// TIA Portal project "Rectz" (V13)

(* hardware
DEVICE "S7300/ET200M station_1"  S7-300 station
   slot 0: "Rail_0"  Rail  6ES7 390-1***0-0AA0
   slot 1: "PS 307 5A_1"  PS 307 5A  6ES7 307-1EA01-0AA0
   slot 2: "PLC_1"  CPU 314C-2 PN/DP  6ES7 314-6EH04-0AB0  V3.3
      slot 2: "PROFINET interface_1"  PN-IO
         slot 1: "Port_1"  Port
         slot 2: "Port_2"  Port
      slot 5: "DI 24/DO 16_1"  DI24/DO16
      slot 6: "AI 5/AO 2_1"  AI5/AO2
      slot 7: "Count_1"  Counter
      slot 8: "Positioning_1"  Positioning
*)

// ===== PLC "PLC_1"  CPU 314C-2 PN/DP =====

VAR_GLOBAL   // PLC tag table "Default tag table"
   "Start" AT %I0.1 : Bool;   // Botão de start
   "Reset" AT %I0.2 : Bool;   // Botão de reset
   "Stop" AT %I0.3 : Bool;   // Botão de stop
   "Emergency stop" AT %I0.4 : Bool;   // Botão de emergência
   "Auto" AT %I0.5 : Bool;   // Chave em estado automático
   "At exit" AT %I0.0 : Bool;   // Sensor retrorreflexivo
   "Entry conveyor" AT %Q0.0 : Bool;   // Esteira de entrada
   "Exit conveyor" AT %Q0.2 : Bool;   // Esteira de sáida
   "flag" AT %M0.0 : Bool;
   "erro" AT %MW2 : Word;
   "Soft 1 belt" AT %Q0.4 : Bool;   // Esteira 1 que empurra os produtos
   "Soft 1 turn" AT %Q0.3 : Bool;   // Esteira 1 gira
   "Soft 2 belt" AT %Q0.6 : Bool;   // Esteira 2 que empurra os produtos
   "Soft 2 turn" AT %Q0.5 : Bool;   // Esteira 2 gira
   "Soft 3 belt" AT %Q1.0 : Bool;   // Esteira 3 que empurra os produtos
   "Soft 3 turn" AT %Q0.7 : Bool;   // Esteira 3 gira
   "s_digital" AT %MD4 : Real;
   "Stop blade" AT %Q0.1 : Bool;
   "Start light" AT %Q1.1 : Bool;   // Led verde do botão start
   "Reset light" AT %Q1.2 : Bool;   // Led amarelo do botão reset
   "Stop light" AT %Q1.3 : Bool;   // Led vermelho do botão stop
   "Vision sensor(1)" AT %I0.7 : Bool;
   "Vision sensor(2)" AT %I1.0 : Bool;
   "Vision sensor(3)" AT %I1.1 : Bool;
   "Vision sensor(4)" AT %I1.2 : Bool;
   "liga_contador" AT %Q1.4 : Bool;
   "memoria" AT %MW8 : Int;
   "desliga_esteira1" AT %Q1.5 : Bool;
   "memoria1" AT %MD10 : Time;
   "desliga_braço1" AT %Q1.6 : Bool;
   "Remover 1" AT %Q1.7 : Bool;
   "Remover 2" AT %Q2.0 : Bool;
   "Remover 3" AT %Q2.1 : Bool;
END_VAR

ORGANIZATION_BLOCK "Main"   // OB1, LAD
TITLE = "Main Program Sweep (Cycle)"
{ S7_Optimized_Access := 'FALSE' }
VERSION : 0.1
   VAR_TEMP
      OB1_EV_CLASS : Byte;   // Bits 0-3 = 1 (Coming event), Bits 4-7 = 1 (Event class 1)
      OB1_SCAN_1 : Byte;   // 1 (Cold restart scan 1 of OB 1), 3 (Scan 2-n of OB 1)
      OB1_PRIORITY : Byte;   // Priority of OB Execution
      OB1_OB_NUMBR : Byte;   // 1 (Organization block 1, OB1)
      OB1_RESERVED_1 : Byte;   // Reserved for system
      OB1_RESERVED_2 : Byte;   // Reserved for system
      OB1_PREV_CYCLE : Int;   // Cycle time of previous OB1 scan (milliseconds)
      OB1_MIN_CYCLE : Int;   // Minimum cycle time of OB1 (milliseconds)
      OB1_MAX_CYCLE : Int;   // Maximum cycle time of OB1 (milliseconds)
      OB1_DATE_TIME : Date_And_Time;   // Date and time OB1 started
   END_VAR
BEGIN
END_ORGANIZATION_BLOCK